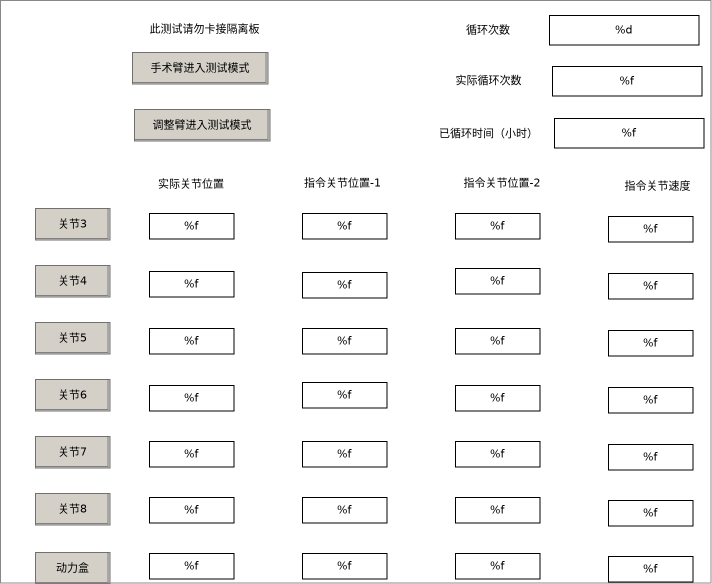
VISUALIZATION arm3CycleTest  // 712x584
VAR_IN_OUT
	
END_VAR
VAR CONSTANT
	arm : INT := 3;
END_VAR
    Button (132,52 136x32), "手术臂进入测试模式", colour toggle: g_cycleTest.m_enterCycleTestMode[3]
        toggle g_cycleTest.m_enterCycleTestMode[3]
    Rectangle (549,15 150x30), "%d", text variable: g_cycleTest.m_targetCycleNum[3]
    Label (446,15 84x30), "循环次数"
    Label (283,169 119x28), "指令关节位置-1"
    Label (141,169 100x30), "实际关节位置"
    Rectangle (149,385 85x26), "%f", text variable: g_systemInfo.m_slaveJntInfo[3,1].m_curJntPos
    Rectangle (149,441 85x26), "%f", text variable: g_systemInfo.m_slaveJntInfo[3,2].m_curJntPos
    Rectangle (149,497 85x26), "%f", text variable: g_systemInfo.m_slaveJntInfo[3,3].m_curJntPos
    Rectangle (149,553 85x26), "%f", text variable: g_systemInfo.m_slaveJntInfo[3,4].m_curJntPos
    Rectangle (149,213 85x26), "%f", text variable: g_systemInfo.m_setupJntInfo[3,3].m_curJntPos
    Rectangle (149,271 85x26), "%f", text variable: g_systemInfo.m_setupJntInfo[3,4].m_curJntPos
    Rectangle (149,328 85x26), "%f", text variable: g_systemInfo.m_setupJntInfo[3,5].m_curJntPos
    Rectangle (302,213 85x26), "%f", text variable: g_cycleTest.m_targetJntPosSetup[3,1][3]
        OnMouseClick: write the text variable via Default
    Rectangle (302,272 85x26), "%f", text variable: g_cycleTest.m_targetJntPosSetup[3,1][4]
        OnMouseClick: write the text variable via Default
    Rectangle (302,328 85x26), "%f", text variable: g_cycleTest.m_targetJntPosSetup[3,1][5]
        OnMouseClick: write the text variable via Default
    Rectangle (302,382 85x26), "%f", text variable: g_cycleTest.m_targetJntPos[3,1][1]
        OnMouseClick: write the text variable via Default
    Rectangle (302,441 85x26), "%f", text variable: g_cycleTest.m_targetJntPos[3,1][2]
        OnMouseClick: write the text variable via Default
    Rectangle (302,497 85x26), "%f", text variable: g_cycleTest.m_targetJntPos[3,1][3]
        OnMouseClick: write the text variable via Default
    Rectangle (302,553 85x26), "%f", text variable: g_cycleTest.m_targetJntPos[3,1][4]
        OnMouseClick: write the text variable via Default
    Label (444,169 116x28), "指令关节位置-2"
    Rectangle (455,213 85x26), "%f", text variable: g_cycleTest.m_targetJntPosSetup[3,2][3]
        OnMouseClick: write the text variable via Default
    Rectangle (455,268 85x26), "%f", text variable: g_cycleTest.m_targetJntPosSetup[3,2][4]
        OnMouseClick: write the text variable via Default
    Rectangle (455,328 85x26), "%f", text variable: g_cycleTest.m_targetJntPosSetup[3,2][5]
        OnMouseClick: write the text variable via Default
    Rectangle (455,385 85x26), "%f", text variable: g_cycleTest.m_targetJntPos[3,2][1]
        OnMouseClick: write the text variable via Default
    Rectangle (455,441 85x26), "%f", text variable: g_cycleTest.m_targetJntPos[3,2][2]
        OnMouseClick: write the text variable via Default
    Rectangle (455,497 85x26), "%f", text variable: g_cycleTest.m_targetJntPos[3,2][3]
        OnMouseClick: write the text variable via Default
    Rectangle (455,553 85x26), "%f", text variable: g_cycleTest.m_targetJntPos[3,2][4]
        OnMouseClick: write the text variable via Default
    Button (134,109 136x32), "调整臂进入测试模式", colour toggle: g_cycleTest.m_enterCycleTestModeSetup[3]
        toggle g_cycleTest.m_enterCycleTestModeSetup[3]
    Label (603,172 109x28), "指令关节速度"
    Rectangle (608,216 85x26), "%f", text variable: g_cycleTest.m_targetJntVelSetup[3][3]
        OnMouseClick: write the text variable via Default
    Rectangle (608,273 85x26), "%f", text variable: g_cycleTest.m_targetJntVelSetup[3][4]
        OnMouseClick: write the text variable via Default
    Rectangle (608,330 85x26), "%f", text variable: g_cycleTest.m_targetJntVelSetup[3][5]
        OnMouseClick: write the text variable via Default
    Rectangle (608,387 85x26), "%f", text variable: g_cycleTest.m_targetJntVelSlave[3][1]
        OnMouseClick: write the text variable via Default
    Rectangle (608,444 85x26), "%f", text variable: g_cycleTest.m_targetJntVelSlave[3][2]
        OnMouseClick: write the text variable via Default
    Rectangle (608,500 85x26), "%f", text variable: g_cycleTest.m_targetJntVelSlave[3][3]
        OnMouseClick: write the text variable via Default
    Rectangle (608,556 85x26), "%f", text variable: g_cycleTest.m_targetJntVelSlave[3][4]
        OnMouseClick: write the text variable via Default
    Rectangle (552,66 150x30), "%f", text variable: g_cycleTest.m_curCycleNum[3]
        OnMouseClick: write the text variable via Default
    Label (440,70 97x21), "实际循环次数"
    Rectangle (554,118 150x30), "%f", text variable: g_cycleTest.m_curCycleTime[3]
        OnMouseClick: write the text variable via Default
    Label (428,123 121x21), "已循环时间（小时）"
    Button (35,208 75x32), "关节3", colour toggle: g_cycleTest.m_disableSetupJntMotion[3][3]
        toggle g_cycleTest.m_disableSetupJntMotion[3][3]
    Button (35,265 75x32), "关节4", colour toggle: g_cycleTest.m_disableSetupJntMotion[3][4]
        toggle g_cycleTest.m_disableSetupJntMotion[3][4]
    Button (35,322 75x32), "关节5", colour toggle: g_cycleTest.m_disableSetupJntMotion[3][5]
        toggle g_cycleTest.m_disableSetupJntMotion[3][5]
    Button (35,379 75x32), "关节6", colour toggle: g_cycleTest.m_disableSlaveJntMotion[3][1]
        toggle g_cycleTest.m_disableSlaveJntMotion[3][1]
    Button (35,436 75x32), "关节7", colour toggle: g_cycleTest.m_disableSlaveJntMotion[3][2]
        toggle g_cycleTest.m_disableSlaveJntMotion[3][2]
    Button (35,493 75x32), "关节8", colour toggle: g_cycleTest.m_disableSlaveJntMotion[3][3]
        toggle g_cycleTest.m_disableSlaveJntMotion[3][3]
    Button (35,552 75x32), "动力盒", colour toggle: g_cycleTest.m_disableSlaveJntMotion[3][4]
        toggle g_cycleTest.m_disableSlaveJntMotion[3][4]
    Label (128,14 153x30), "此测试请勿卡接隔离板"
END_VISUALIZATION

(* stored: Version 1.1.0.1, ProductVersion 3.1.4024.11
   Visu arm3CycleTest: Id {a06bd5ac-0f46-43b6-b689-0c090f3de4db} *)
